# B&R Automation Studio project TestMappView
Automation Studio 4.7.6.114 SP; technology packages: mapp 5.15.0, mappView 5.15.1

## Configuration Config1

CPU PC_any, AutomationRuntime C4.72, Build 4.1.2, Safety 0.0, Vc V4.72.0

### Task classes (Cpu.sw)
```
Cyclic#4:
  MainProgra <- MainProgram.prg
  TestMotor <- TestMotor.prg
  Alarm <- Alarm.prg
Libraries: MTBasics, brsystem, MTTypes, sys_lib, runtime, Library, MpServer, MpAlarmX, MpBase, astime
```

### Hardware
```
PC : PC_any v1.1.0.0 (OrderNumber=PC)
  ConfigurationID = TestMappView_Config1
  ActivateOpcUa = 1
  OpcUaInformationModels_PV_Version = 1
```

### Config.mpalarmxcore - PC/mappServices/Config.mpalarmxcore
```
Element gAlarmXCore (Type=mpalarmxcore)
  mapp.AlarmX.Core:
    BySeverity:
      [0]:
        Severity = 1
        [0] = Reaction
          Name = InfoActive
  mapp.AlarmX.Core.Configuration:
    [0]:
      Name = Alarm1
      Message = Alarm 1  {=$AlarmTexts/{&snippet1}}
    [1]:
      Name = Alarm2
      Message = Alarm 2 is active
      Severity = 11
      Behavior = PersistentAlarm
    [2]:
      Name = d
  mapp.AlarmX.Core.Snippets:
    [0]:
      Key = snippet1
      Value:
        PV = ::Alarm:snippet1
  mapp.AlarmX.Core.Categories:
    [0]:
      Name = Information
      SourceProperty:
        Severity = 1
```

### Config_1.mpalarmxhistory - PC/mappServices/Config_1.mpalarmxhistory
```
Element gAlarmXHistory (Type=mpalarmxhistory)
  mapp.AlarmX.History:
    Memory:
      MemorySize = 500
      MemoryType = 0
```

## Logical view

Binary libraries used (declarations not repeated): operator, runtime, astime, AsIecCon, MTBasics 5.06.0, brsystem, MTTypes 1.03.4, sys_lib, MpServer 5.15.0, MpAlarmX 5.15.0, MpBase 5.15.0

### Global.typ - Globale Datentypen
```iecst
TYPE
	ClientInfoType : 	STRUCT
		BrowseResolution : WSTRING[80];
		LanguageId : WSTRING[3];
		SlotId : SINT;
		IpAddress : WSTRING[15];
		IsValid : BOOL;
		UserId : WSTRING[80];
	END_STRUCT;

	TestEnum :
	(
		One,
		Two
	);

	TestEnum2 :
		(
		One2,
		Two2
	);
END_TYPE
```

### Global.var - Globale Variablen
```iecst
VAR
	testInt : INT;
	ClientInfo : ARRAY[0..2] OF ClientInfoType;

	gIstTemp : INT;
	gSollTemp : INT;

	gDropDownItems : ARRAY[0..2] OF STRING[100];
	gDropDownSelectedValue : STRING[100];
	gDropDownSelectedIndex : INT;
	gIntFromString : INT;

END_VAR
```

### Package Logical/Libraries - Globale Bibliotheken

- Visualisation Logical/mappView (not shown)

### Program Logical/MainProgram (IEC)

#### Main.st - Init, cyclic, exit code
```iecst
PROGRAM _INIT
	(* Insert code here *)
	 gSollTemp := 25;
END_PROGRAM

PROGRAM _CYCLIC
	(* Insert code here *)
	MTBasicPT1.Enable := TRUE;
	MTBasicPT1.Gain := 1;
	MTBasicPT1.TimeConstant := 1;
	MTBasicPT1.In := INT_TO_REAL(gSollTemp);
	MTBasicPT1();

	gIstTemp := REAL_TO_INT(MTBasicPT1.Out);

	ClientInfo;

	// Test Drop Down
	gDropDownItems;
	gDropDownSelectedIndex;
	gDropDownSelectedValue;

	gIntFromString := STRING_TO_INT(gDropDownSelectedValue);

	(*******************************************************************
	* Test Style Change
	*
	*******************************************************************)

	visuChangeStyleFromWidget;

	visuStyle;

END_PROGRAM

PROGRAM _EXIT
	(* Insert code here *)

END_PROGRAM
```

#### Variables.var - Local variables
```iecst
VAR
	MTBasicPT1 : MTBasicsPT1;
	visuChangeStyleFromWidget : BOOL;
	visuStyle : STRING;
END_VAR
```

### Program Logical/Alarm (IEC)

#### Cyclic.st - Cyclic code
```iecst
PROGRAM _CYCLIC
	(* Insert code here *)

	//Call Alarm Handler
	FB_MpAlarmXCore(
		MpLink := ADR(gAlarmXCore),
		Enable := TRUE,
		ErrorReset := cmdErrorReset);

	//Call Alarm History Handler
	FB_MpAlarmXHistory(
		MpLink := ADR(gAlarmXHistory),
		Enable := TRUE,
		ErrorReset := cmdErrorReset,
		DeviceName := ADR('CF'));

	//Edge Alarme
	IF cmdAlarm1 THEN
		snippet1 := 1;
		MpAlarmXSet(gAlarmXCore, 'Alarm1');

		snippet1 := 2;
		MpAlarmXSet(gAlarmXCore, 'Alarm1');

		snippet1 := 3;
		MpAlarmXSet(gAlarmXCore, 'Alarm1');

		cmdAlarm1 := FALSE;
	END_IF;

	//Perm
	IF cmdAlarm2 THEN
		cmdAlarm2 := FALSE;
		MpAlarmXSet(gAlarmXCore, 'Alarm2');

	END_IF;

	IF resetAlarm2 THEN
		resetAlarm2 := FALSE;
		MpAlarmXReset(gAlarmXCore, 'Alarm2');
	END_IF;

	FB_AlarmResetAll(
		MpLink := ADR(gAlarmXCore),
		Enable := TRUE,
		ErrorReset := cmdErrorReset,
		Execute := cmdErrorReset);

	cmdErrorReset := FALSE;

	snippet1;

END_PROGRAM
```

#### Variables.var - Local variables
```iecst
VAR

	FB_MpAlarmXCore : MpAlarmXCore;
	FB_MpAlarmXHistory : MpAlarmXHistory;
	FB_AlarmResetAll : MpAlarmXAcknowledgeAll;
	cmdErrorReset : BOOL;
	cmdAlarm1 : BOOL;
	cmdAlarm2 : BOOL;
	cmdAlarm3 : BOOL;
	resetAlarm1 : BOOL;
	resetAlarm2 : BOOL;
	resetAlarm3 : BOOL;
	snippet1 : USINT;
	snippet2 : USINT;
	snippet3 : USINT;

END_VAR
```

### Program Logical/TestMotor (IEC)

#### Main.st - Init, cyclic, exit code
```iecst
(********************************************************************
 * COPYRIGHT -- MIEtech GmbH & Co. KG
 ********************************************************************
 * Program:	TestMotor
 * File:	Main.st
 * Author:	D.Graf
 * Created:	01.10.2021
 * Changed:	05.01.2020, MM, example changelog discription 1
 *			20.10.2021, DG, Add Motor Functions
 ********************************************************************
 * Motor Program
 ********************************************************************)

PROGRAM _INIT
	(* Insert code here *)

END_PROGRAM

PROGRAM _CYCLIC
	(* Insert code here *)

END_PROGRAM

PROGRAM _EXIT
	(* Insert code here *)

END_PROGRAM
```

#### Variables.var - Local variables
```iecst
VAR

	ready : BOOL;
	motorIsReady : BOOL;

	FbMotor1 : FB_Motor;
	FbMotoren : ARRAY[1..2] OF FB_Motor;

END_VAR
```

#### MotorActions.st
```iecst
ACTION ActionMotor:

END_ACTION

ACTION NewAction :
	(* Insert code here *)

END_ACTION
```

### Library Logical/Library (IEC)

#### Types.typ - Exported data types
```iecst
TYPE
	Type_MotorParameter : 	STRUCT
		Param1 : BOOL;
		Param2 : USINT;
	END_STRUCT;
	Type_MotorCommand : 	STRUCT
		CMD1 : BOOL;
		CMD2 : USINT;
	END_STRUCT;
	Type_Motor : 	STRUCT
		Param : Type_MotorParameter;
		Cmd : Type_MotorCommand;
	END_STRUCT;
END_TYPE
```

#### Library.fun - Exported functions and function blocks
```iecst
FUNCTION_BLOCK FB_Motor
	VAR_INPUT
		Enable : BOOL;
		Cmd : Type_MotorCommand;
		Parameter : Type_MotorParameter;
	END_VAR
	VAR_OUTPUT
		Status : USINT;
	END_VAR
	VAR_IN_OUT
		ErrorCounter : USINT;
	END_VAR
	VAR
		step : USINT;
	END_VAR
END_FUNCTION_BLOCK
```

#### FB_Motor.st
```iecst
(**************************************************************************************************************
* COPYRIGHT -- MIEtech GmbH & CO. KG
**************************************************************************************************************
* FB:		FB_Motor
* File:		FB_Motor.st
* Author:	D.Graf
* Created:	01.10.2021
**************************************************************************************************************
* Description:
*			This function block deals with the control of a simple motor
*
**************************************************************************************************************
* ChangeLog:
*			18.10.2021, MM, example changelog discription 1
*			20.10.2021, DG, Add new Function XY
**************************************************************************************************************)

FUNCTION_BLOCK FB_Motor
	IF Enable THEN
		// Main Code

	ELSE
		//z.B.: Reset all Signals
		// Set Status to Not Enable or else

	END_IF;

END_FUNCTION_BLOCK
```

Listed in the project but not available here: Logical/MainProgram/Types.typ, Logical/Alarm/Init.st, Logical/Alarm/Exit.st, Logical/TestMotor/Types.typ, Logical/Library/Constants.var
